# EPICS autosave request: iocBoot/ioc13laser/auto_settings.req
file "scan_settings.req",               P=$(P), S=scan1
file "scan_settings.req",               P=$(P), S=scan2
file "scan_settings.req",               P=$(P), S=scan3
file "scan_settings.req",               P=$(P), S=scan4
file "CARS_8_motor_settings.req",       P=$(P)
